{attribute 'linkalways'} 
{attribute 'no_explicit_call' := 'This FB is a CLASS and must be accessed using methods or properties'}
{attribute 'enable_dynamic_creation'}
FUNCTION_BLOCK _SINT EXTENDS NumericDatatypeBase
VAR
	localData : SINT;
	activeData : REFERENCE TO SINT REF= localData;
END_VAR

PROPERTY PUBLIC Address : PVOID
GET
Address := ADR(activeData);
END_GET
END_PROPERTY

METHOD PUBLIC ClearReference
VAR_INPUT
END_VAR
activeData REF= localData;
END_METHOD

METHOD PUBLIC Clone : I_Datatype
VAR
    pClone : POINTER TO _SINT;
END_VAR
pClone := __NEW(_SINT(InitialValue := Value));
Clone := pClone^;
END_METHOD

METHOD FB_init : BOOL
VAR_INPUT
	bInitRetains : BOOL; // if TRUE, the retain variables are initialized (warm start / cold start)
	bInCopyCode : BOOL;  // if TRUE, the instance afterwards gets moved into the copy code (online change)
	InitialValue : SINT;
END_VAR
localData := InitialValue;
END_METHOD

PROPERTY PUBLIC IsFloat : BOOL
GET
IsFloat := FALSE;
END_GET
END_PROPERTY

PROPERTY PUBLIC IsSigned : BOOL
GET
IsSigned := TRUE;
END_GET
END_PROPERTY

METHOD PUBLIC MakeReferenceTo
VAR_INPUT
	ReferenceTarget : REFERENCE TO SINT;
END_VAR
activeData REF= ReferenceTarget;
END_METHOD

PROPERTY PUBLIC MaxValue : SINT
GET
MaxValue :=  DatatypeLimits.SINT_MAX_VALUE;
END_GET
END_PROPERTY

PROPERTY PUBLIC MinValue : SINT
GET
MinValue := DatatypeLimits.SINT_MIN_VALUE;
END_GET
END_PROPERTY

METHOD PROTECTED SerializeMaxValue
VAR_INPUT
	Serializer : I_Serializer;
END_VAR
Serializer.AddSint(MaxValue);
END_METHOD

METHOD PROTECTED SerializeMinValue
VAR_INPUT
	Serializer : I_Serializer;
END_VAR
Serializer.AddSint(MinValue);
END_METHOD

METHOD PUBLIC SerializeWith
VAR_INPUT
	Serializer : I_Serializer;
END_VAR
Serializer.AddSint(activeData);
END_METHOD

PROPERTY PUBLIC Size : UDINT
GET
Size := SIZEOF(activeData);
END_GET
END_PROPERTY

METHOD TryDeserializeFrom : BOOL
VAR_INPUT
	Deserializer : I_Deserializer;
	Feedback : I_DeserializerFeedback;
END_VAR
TryDeserializeFrom := Deserializer.TryGetSint(activeData, Feedback);
END_METHOD

METHOD TryMakeReferenceTo : BOOL
VAR_INPUT
	Target : I_Datatype;
END_VAR
VAR
	pTargetData : POINTER TO SINT;
END_VAR
IF NOT (Target.TypeName = TypeName) THEN
	RETURN;
END_IF

pTargetData := Target.Address;
activeData REF= pTargetData^;
TryMakeReferenceTo := TRUE;
END_METHOD

PROPERTY PUBLIC TypeName : T_MAXSTRING
GET
TypeName := 'SINT';
END_GET
END_PROPERTY

PROPERTY PUBLIC Value : REFERENCE TO SINT
GET
Value REF= activeData;
END_GET
END_PROPERTY

END_FUNCTION_BLOCK

(* stored: Version 1.1.0.1, ProductVersion 3.1.4024.12
   POU _SINT: Id {122dae3f-1273-407a-bdae-00ea5e1a351a}, SpecialFunc None
   Folder Constructor: Id {620d8041-d200-494e-a9ed-e17e20d816fc}
   Folder Protected: Id {49ec95fa-b67e-47c5-8f75-69b18b64e960}
   Property Address: Id {4ddd0566-0a63-4e49-9352-cc96c83081a4}
   Get Get: Id {96b793ff-234d-4067-91dc-7cfdf170fbc7}
   Method ClearReference: Id {dd773684-6d6f-42d9-b0f6-37fbc077f9e4}
   Method Clone: Id {7049dd9b-4aeb-46ba-a2de-729447d77a3f}
   Method FB_init: Id {e7aab2c8-9995-47db-a1c1-cb95393376c4}
   Property IsFloat: Id {2560d36f-245d-4358-86f0-416fcd4ec702}
   Get Get: Id {d20517ba-96cd-416f-812c-1a43495aa00a}
   Property IsSigned: Id {727e2535-e220-494b-a91a-2d750f420fda}
   Get Get: Id {4992e98b-018a-46ab-a2e9-65e69df1ec4d}
   Method MakeReferenceTo: Id {01a4a022-49ba-4f1b-8d8f-931d313003c5}
   Property MaxValue: Id {1695e1cb-46ec-45b5-b736-7d31692ea918}
   Get Get: Id {52db4707-d80f-4974-bb04-59210d9e22e8}
   Property MinValue: Id {65e7ba36-6d34-48c4-90cf-358f31d16e5d}
   Get Get: Id {2a127439-4478-4a63-a6b3-7e84bf6f4035}
   Method SerializeMaxValue: Id {cefeec5e-1261-4fc3-8a96-0f583754b051}
   Method SerializeMinValue: Id {2d0abd04-e5ed-4897-a9f7-b546e3623d1d}
   Method SerializeWith: Id {68ba6099-8e9c-4cb6-b8be-a3cf464e9e1b}
   Property Size: Id {d6e1d4df-d1c1-4de1-9586-d1b9aff0e0a0}
   Get Get: Id {b8e1e8f0-5f8c-40d7-9646-7c5c99df1d92}
   Method TryDeserializeFrom: Id {5cd18f75-5029-48ea-8dad-a46f1b9b3e2d}
   Method TryMakeReferenceTo: Id {c3f6a5d7-9307-460c-a89a-e3ce28f84912}
   Property TypeName: Id {ce884252-29b0-459b-b0c7-c78add9ed838}
   Get Get: Id {aa939f2f-2a9d-4703-ac26-e1ad2269cf20}
   Property Value: Id {ba767074-e750-4e97-97b2-95346054af2d}
   Get Get: Id {8221e489-838c-452c-bc29-60cb7f7f8afb} *)
